INTERFACE I_FourStateDevice

METHOD Off
VAR_INPUT
END_VAR
END_METHOD

METHOD On
VAR_INPUT
END_VAR
END_METHOD

METHOD State_1
VAR_INPUT
END_VAR
END_METHOD

METHOD State_2
VAR_INPUT
END_VAR
END_METHOD

METHOD State_3
VAR_INPUT
END_VAR
END_METHOD

METHOD State_4
VAR_INPUT
END_VAR
END_METHOD

PROPERTY Status : INT
GET
END_GET
END_PROPERTY

END_INTERFACE

(* stored: Version 1.1.0.1, ProductVersion 3.1.4024.13
   Itf I_FourStateDevice: Id {8d4d81c2-0104-4c46-9a2d-913dc4a57210}
   Method Off: Id {18457cd9-8db7-400e-ae3d-73e768dc029a}
   Method On: Id {8d8d8e76-9862-4573-a2a8-e120dc926f9c}
   Method State_1: Id {1397b85e-5982-4a76-b821-afba878c6f2c}
   Method State_2: Id {9385268f-4882-4ab2-bd91-812ae810fee3}
   Method State_3: Id {2bfbb433-0a97-4640-b740-1ce42e5f1890}
   Method State_4: Id {9adb5188-1389-4291-9c34-0c4365c839c2}
   Property Status: Id {e1c08cd5-1904-4910-8f25-b0cc92be0cd4}
   Get Get: Id {8df65787-5010-4baa-a176-26f47f000ad1} *)
